Yaskawa INFORM job: IN-TUNNEL.JBI

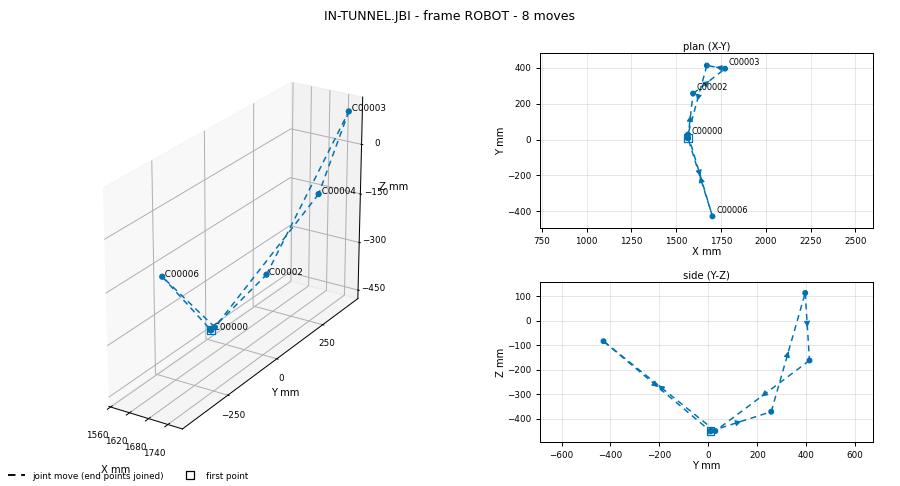
[picture p0: tool path of IN-TUNNEL.JBI in frame ROBOT, 8 of 8 moves have a stored position in this frame; points joined in program order, loops and branches not executed]
/JOB
//NAME IN-TUNNEL
///FOLDERNAME IMPORTANT_JOBS
//POS
///NPOS 8,8,0,0,0,0
///TOOL 0
///POSTYPE ROBOT
///RECTAN
///RCONF 1,0,1,0,0,0,0,0,0,0,0,0,0,0,0,0,0,0,0,0,0,0,0,0
C00000=1565.876,8.473,-450.584,0.8006,-14.6203,-0.0454
C00001=1565.876,8.473,-450.584,0.8006,-14.6203,-0.0454
C00002=1594.520,256.653,-371.064,34.1867,-8.6914,-19.6119
C00003=1773.118,395.447,114.208,96.9926,29.3892,-37.0963
C00004=1671.343,413.011,-161.605,64.9806,7.1387,-33.2097
C00005=1566.114,28.264,-449.788,3.3561,-14.5779,-1.6020
C00006=1702.675,-428.515,-82.947,-74.2121,14.0741,36.1483
C00007=1565.876,8.473,-450.584,0.8006,-14.6203,-0.0454
///RCONF 0,0,0,0,0,0,0,0,0,0,0,0,0,0,0,0,0,0,0,0,0,0,0,0
BC00000=3362.479
BC00001=5704.936
BC00002=5704.936
BC00003=5704.936
BC00004=5704.936
BC00005=5704.936
BC00006=5704.936
BC00007=3362.479
//INST
///DATE 2024/04/16 08:57
///ATTR SC,RW,RJ
////FRAME ROBOT
///GROUP1 RB1,BS1
NOP
MOVJ C00000 BC00000 VJ=30.00
MOVJ C00001 BC00001 VJ=30.00
MOVJ C00002 BC00002 VJ=30.00
MOVJ C00003 BC00003 VJ=30.00
TIMER T=0.50
MOVJ C00004 BC00004 VJ=30.00
MOVJ C00005 BC00005 VJ=30.00
MOVJ C00006 BC00006 VJ=30.00
TIMER T=0.50
MOVJ C00007 BC00007 VJ=30.00
END
